Universal Robots PolyScope program: RuchL1MS.urp

Program RuchL1MS (installation=default directory=/programs/usbdisk createdIn=3.15.8.106339 lastSavedIn=3.15.8.106339 robotSerialNumber=2020330428)
Calibrated DH parameters: a=[0.000029, -0.241913, -0.128453, -0.000049, -0.000012, 0]; d=[0.151842, -4.082088, 33.504745, -29.309875, 0.08529, 0.082285]; alpha=[1.571059, -0.006644, 0.005794, 1.571984, -1.571997, 0]; deltaTheta=[-0.000032, 0.111537, 0.813391, -0.924919, 0.000036, 0.000016]
Robot Program (runOnlyOnce=false)
  MoveL speed 200 mm/s, acceleration 400 mm/s^2 (useActiveTCP=true) feature=Base
    Waypoint Punkt_orienta_3: TCP in base x=236.723 y=-112.694 z=87.696 mm, rx=2.2254 ry=-2.2101 rz=0.0056 rad; joints [0, -90, -135, -45, 90, 0] deg; flange x=236.81 y=-112.23 z=162.695 mm, rx=2.2254 ry=-2.2101 rz=0.0056 rad
    Waypoint Punkt_orienta_4: TCP in base x=236.199 y=-111.927 z=388.816 mm, rx=2.2233 ry=-2.2188 rz=-0.0017 rad; joints [0.004, -89.999, -45, -135, 90, 0.002] deg; flange x=236.288 y=-111.954 z=463.816 mm, rx=2.2233 ry=-2.2188 rz=-0.0017 rad
